_CFC_ (* Continuous Function Chart, elements in execution order *)
#0 INT_TO_REAL(SHU6_PV1_1TE3_AI3)
#1 DIV(#0, 10)
#2 SHU6_PV1_TE3_VN <= #1
#3 I_GT_TE:ISTOK_GT(dost: TRUE, x: #1, ust: SHU6_PV1_TE_HIGHLIMIT, shkal: -, gist: 1)
#4 I_LT_TE:ISTOK_LT(dost: TRUE, x: #1, ust: SHU6_PV1_TE_LOWLIMIT, shkal: -, gist: 1)
#5 OR(#3.Xb, #4.Xm)
#6 TON_DOST:TON(IN: NOT #5, PT: T#10s)
#7 SHU6_PV1_TE3_DOST <= #6.Q
#8 SUB(SHU6_PV1_TE3_T_UST, 0.6)
#9 fb_TE3_M_UST:ISTOK_LT(dost: #6.Q, x: #1, ust: #8, shkal: -, gist: 0.5)
#10 SHU6_PV1_TE3_M_UST <= #9.Xm
#11 SHU6_PV1_TE3_NM_UST <= #9.XmN
#12 ADD(SHU6_PV1_TE3_T_UST, 0.6)
#13 fb_TE3_B_UST:ISTOK_GT(dost: #6.Q, x: #1, ust: #12, shkal: -, gist: 0.5)
#14 SHU6_PV1_TE3_B_UST <= #13.Xb
#15 SHU6_PV1_TE3_NB_UST <= #13.XbN
_END_CFC_
(* the same logic as Structured Text *)
_t47 := INT_TO_REAL(SHU6_PV1_1TE3_AI3) / 10;
SHU6_PV1_TE3_VN := _t47;
I_GT_TE(dost := TRUE, x := _t47, ust := SHU6_PV1_TE_HIGHLIMIT, gist := 1);
I_LT_TE(dost := TRUE, x := _t47, ust := SHU6_PV1_TE_LOWLIMIT, gist := 1);
TON_DOST(IN := NOT (I_GT_TE.Xb OR I_LT_TE.Xm), PT := T#10s);
SHU6_PV1_TE3_DOST := TON_DOST.Q;
fb_TE3_M_UST(dost := TON_DOST.Q, x := _t47, ust := SHU6_PV1_TE3_T_UST - 0.6, gist := 0.5);
SHU6_PV1_TE3_M_UST := fb_TE3_M_UST.Xm;
SHU6_PV1_TE3_NM_UST := fb_TE3_M_UST.XmN;
fb_TE3_B_UST(dost := TON_DOST.Q, x := _t47, ust := SHU6_PV1_TE3_T_UST + 0.6, gist := 0.5);
SHU6_PV1_TE3_B_UST := fb_TE3_B_UST.Xb;
SHU6_PV1_TE3_NB_UST := fb_TE3_B_UST.XbN;
END_PROGRAM

(* POU Input/CI/MRQ1_OB, CFC *)
PROGRAM MRQ1_OB
VAR
	ofset: INT := 0;
	dost_ton_3: TON;
	SR_DOST_MV1: RS;
	fb_MV1b30: ISTOK_GT;
	fb_MV1_OBRb45: ISTOK_GT;
	fb_MV1_OBRm0_1: ISTOK_LT;
	fb_MV1_OBRbSM: ISTOK_GT;
END_VAR
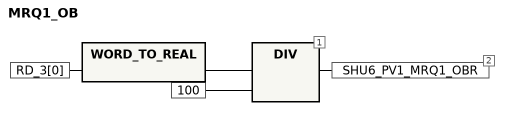
_CFC_ (* Continuous Function Chart, elements in execution order *)
#0 WORD_TO_REAL(RD_3[0])
#1 DIV(#0, 100)
#2 SHU6_PV1_MRQ1_OBR <= #1
_END_CFC_
(* the same logic as Structured Text *)
SHU6_PV1_MRQ1_OBR := WORD_TO_REAL(RD_3[0]) / 100;
END_PROGRAM

(* POU TZBiS/S/ALL_S, CFC *)
PROGRAM ALL_S
VAR
END_VAR
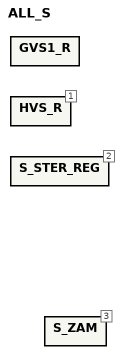
_CFC_ (* Continuous Function Chart, elements in execution order *)
#0 GVS1_R()
#1 HVS_R()
#2 S_STER_REG()
#3 S_ZAM()
_END_CFC_
(* the same logic as Structured Text *)
GVS1_R();
HVS_R();
S_STER_REG();
S_ZAM();
END_PROGRAM

(* POU TZBiS/S/GVS1_R, CFC *)
PROGRAM GVS1_R
VAR
	rs_gvs1: RS;
	GVS1_RUN: BOOL;
END_VAR
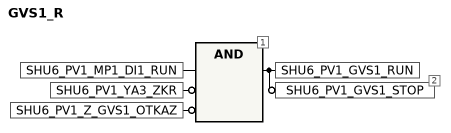
_CFC_ (* Continuous Function Chart, elements in execution order *)
#0 SHU6_PV1_GVS1_RUN <= #1
#1 AND(SHU6_PV1_MP1_DI1_RUN, NOT SHU6_PV1_YA3_ZKR, NOT SHU6_PV1_Z_GVS1_OTKAZ)
#2 SHU6_PV1_GVS1_STOP <= NOT #1
_END_CFC_
END_PROGRAM

(* POU TZBiS/S/HVS_R, CFC *)
PROGRAM HVS_R
VAR
END_VAR
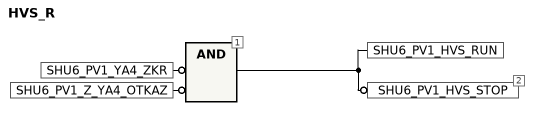
_CFC_ (* Continuous Function Chart, elements in execution order *)
#0 SHU6_PV1_HVS_RUN <= #1
#1 AND(NOT SHU6_PV1_YA4_ZKR, NOT SHU6_PV1_Z_YA4_OTKAZ)
#2 SHU6_PV1_HVS_STOP <= NOT #1
_END_CFC_
END_PROGRAM

(* POU TZBiS/S/S_STER_REG, CFC *)
PROGRAM S_STER_REG
VAR
	ZAD_S_Ster_Reg: TON;
END_VAR
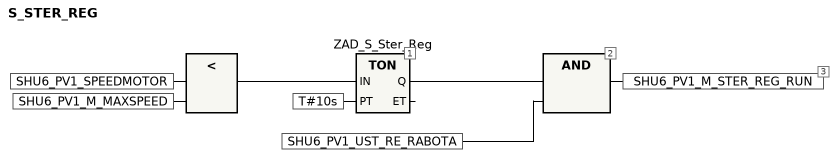
_CFC_ (* Continuous Function Chart, elements in execution order *)
#0 <(SHU6_PV1_SPEEDMOTOR, SHU6_PV1_M_MAXSPEED)
#1 ZAD_S_Ster_Reg:TON(IN: #0, PT: T#10s)
#2 AND(#1.Q, SHU6_PV1_UST_RE_RABOTA)
#3 SHU6_PV1_M_STER_REG_RUN <= #2
_END_CFC_
END_PROGRAM

(* POU TZBiS/S/S_ZAM, CFC *)
PROGRAM S_ZAM
VAR
	SR_ZAM: SR;
END_VAR
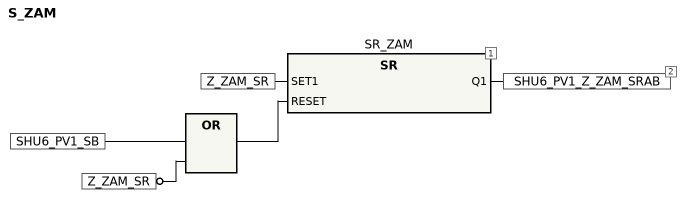
_CFC_ (* Continuous Function Chart, elements in execution order *)
#0 OR(SHU6_PV1_SB, NOT Z_ZAM_SR)
#1 SR_ZAM:SR(SET1: Z_ZAM_SR, RESET: #0)
#2 SHU6_PV1_Z_ZAM_SRAB <= #1.Q1
_END_CFC_
(* the same logic as Structured Text *)
SR_ZAM(SET1 := Z_ZAM_SR, RESET := SHU6_PV1_SB OR NOT Z_ZAM_SR);
SHU6_PV1_Z_ZAM_SRAB := SR_ZAM.Q1;
END_PROGRAM

(* POU TZBiS/TZB/ALL_TZB, CFC *)
PROGRAM ALL_TZB
VAR
END_VAR
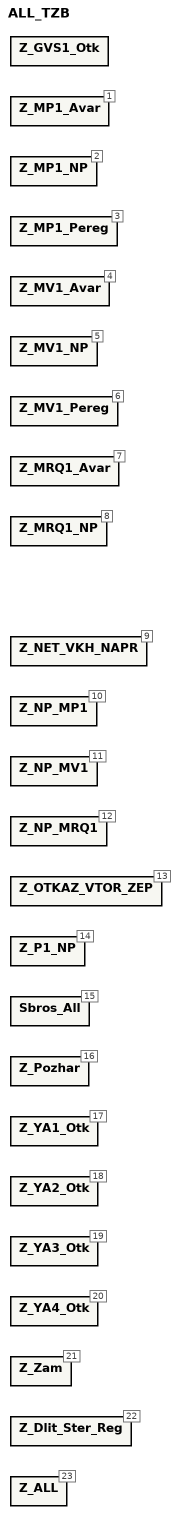
_CFC_ (* Continuous Function Chart, elements in execution order *)
#0 Z_GVS1_Otk()
#1 Z_MP1_Avar()
#2 Z_MP1_NP()
#3 Z_MP1_Pereg()
#4 Z_MV1_Avar()
#5 Z_MV1_NP()
#6 Z_MV1_Pereg()
#7 Z_MRQ1_Avar()
#8 Z_MRQ1_NP()
#9 Z_NET_VKH_NAPR()
#10 Z_NP_MP1()
#11 Z_NP_MV1()
#12 Z_NP_MRQ1()
#13 Z_OTKAZ_VTOR_ZEP()
#14 Z_P1_NP()
#15 Sbros_All()
#16 Z_Pozhar()
#17 Z_YA1_Otk()
#18 Z_YA2_Otk()
#19 Z_YA3_Otk()
#20 Z_YA4_Otk()
#21 Z_Zam()
#22 Z_Dlit_Ster_Reg()
#23 Z_ALL()
_END_CFC_
(* the same logic as Structured Text *)
Z_GVS1_Otk();
Z_MP1_Avar();
Z_MP1_NP();
Z_MP1_Pereg();
Z_MV1_Avar();
Z_MV1_NP();
Z_MV1_Pereg();
Z_MRQ1_Avar();
Z_MRQ1_NP();
Z_NET_VKH_NAPR();
Z_NP_MP1();
Z_NP_MV1();
Z_NP_MRQ1();
Z_OTKAZ_VTOR_ZEP();
Z_P1_NP();
Sbros_All();
Z_Pozhar();
Z_YA1_Otk();
Z_YA2_Otk();
Z_YA3_Otk();
Z_YA4_Otk();
Z_Zam();
Z_Dlit_Ster_Reg();
Z_ALL();
END_PROGRAM

(* POU TZBiS/TZB/Z_GVS1_Otk, CFC *)
PROGRAM Z_GVS1_Otk
VAR
	TON_YA2_OTKAZ: TON;
	SR_GVS1_Otkaz: SR;
	TON_YA2_Z_ZAM: TON;
END_VAR
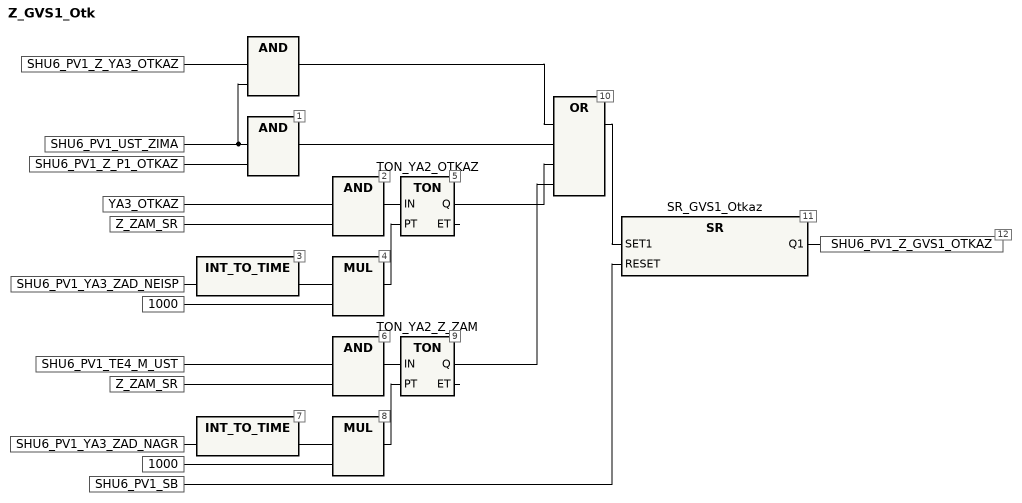
_CFC_ (* Continuous Function Chart, elements in execution order *)
#0 AND(SHU6_PV1_Z_YA3_OTKAZ, SHU6_PV1_UST_ZIMA)
#1 AND(SHU6_PV1_UST_ZIMA, SHU6_PV1_Z_P1_OTKAZ)
#2 AND(YA3_OTKAZ, Z_ZAM_SR)
#3 INT_TO_TIME(SHU6_PV1_YA3_ZAD_NEISP)
#4 MUL(#3, 1000)
#5 TON_YA2_OTKAZ:TON(IN: #2, PT: #4)
#6 AND(SHU6_PV1_TE4_M_UST, Z_ZAM_SR)
#7 INT_TO_TIME(SHU6_PV1_YA3_ZAD_NAGR)
#8 MUL(#7, 1000)
#9 TON_YA2_Z_ZAM:TON(IN: #6, PT: #8)
#10 OR(#0, #1, #5.Q, #9.Q)
#11 SR_GVS1_Otkaz:SR(SET1: #10, RESET: SHU6_PV1_SB)
#12 SHU6_PV1_Z_GVS1_OTKAZ <= #11.Q1
_END_CFC_
(* the same logic as Structured Text *)
TON_YA2_OTKAZ(IN := YA3_OTKAZ AND Z_ZAM_SR, PT := INT_TO_TIME(SHU6_PV1_YA3_ZAD_NEISP) * 1000);
TON_YA2_Z_ZAM(IN := SHU6_PV1_TE4_M_UST AND Z_ZAM_SR, PT := INT_TO_TIME(SHU6_PV1_YA3_ZAD_NAGR) * 1000);
SR_GVS1_Otkaz(SET1 := (SHU6_PV1_Z_YA3_OTKAZ AND SHU6_PV1_UST_ZIMA) OR (SHU6_PV1_UST_ZIMA AND SHU6_PV1_Z_P1_OTKAZ) OR TON_YA2_OTKAZ.Q OR TON_YA2_Z_ZAM.Q, RESET := SHU6_PV1_SB);
SHU6_PV1_Z_GVS1_OTKAZ := SR_GVS1_Otkaz.Q1;
END_PROGRAM

(* POU TZBiS/TZB/Z_MP1_Avar, CFC *)
PROGRAM Z_MP1_Avar
VAR
	SR_MP1_Avar: SR;
	SR_MP2_Avar: SR;
END_VAR
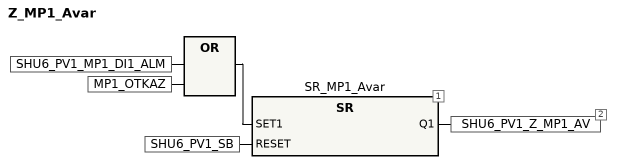
_CFC_ (* Continuous Function Chart, elements in execution order *)
#0 OR(SHU6_PV1_MP1_DI1_ALM, MP1_OTKAZ)
#1 SR_MP1_Avar:SR(SET1: #0, RESET: SHU6_PV1_SB)
#2 SHU6_PV1_Z_MP1_AV <= #1.Q1
_END_CFC_
(* the same logic as Structured Text *)
SR_MP1_Avar(SET1 := SHU6_PV1_MP1_DI1_ALM OR MP1_OTKAZ, RESET := SHU6_PV1_SB);
SHU6_PV1_Z_MP1_AV := SR_MP1_Avar.Q1;
END_PROGRAM

(* POU TZBiS/TZB/Z_MP1_NP, CFC *)
PROGRAM Z_MP1_NP
VAR
	SR_M1_NPit: SR;
	SR_M2_NPit: SR;
END_VAR
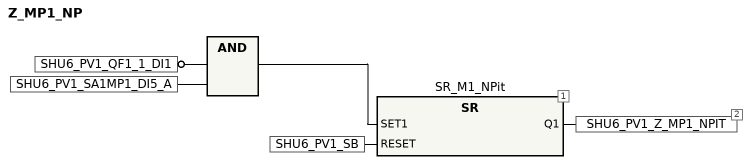
_CFC_ (* Continuous Function Chart, elements in execution order *)
#0 AND(NOT SHU6_PV1_QF1_1_DI1, SHU6_PV1_SA1MP1_DI5_A)
#1 SR_M1_NPit:SR(SET1: #0, RESET: SHU6_PV1_SB)
#2 SHU6_PV1_Z_MP1_NPIT <= #1.Q1
_END_CFC_
(* the same logic as Structured Text *)
SR_M1_NPit(SET1 := NOT SHU6_PV1_QF1_1_DI1 AND SHU6_PV1_SA1MP1_DI5_A, RESET := SHU6_PV1_SB);
SHU6_PV1_Z_MP1_NPIT := SR_M1_NPit.Q1;
END_PROGRAM

(* POU TZBiS/TZB/Z_MP1_Pereg, CFC *)
PROGRAM Z_MP1_Pereg
VAR
	SR_SHU6_PV1_TSMP1_DI4: SR;
	TOF_TSMP1: TOF;
	TON1: TON;
END_VAR
VAR (* helpers for the ST form of the networks *)
	_t23 : BOOL;
END_VAR
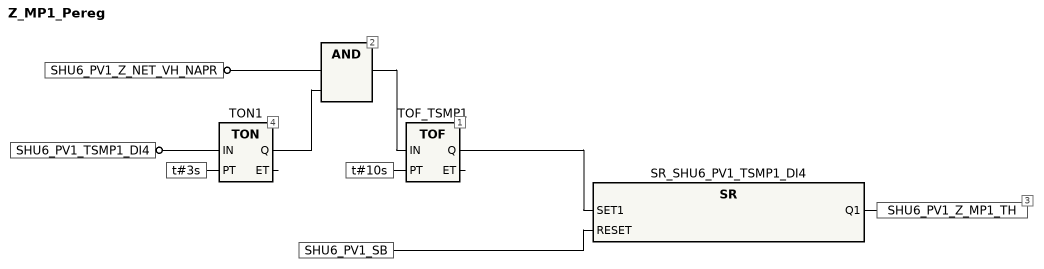
